// Mitsubishi GX Works2 project: 실린더제어ABAB   PLC: Q02/Q02H

PROGRAM MAIN
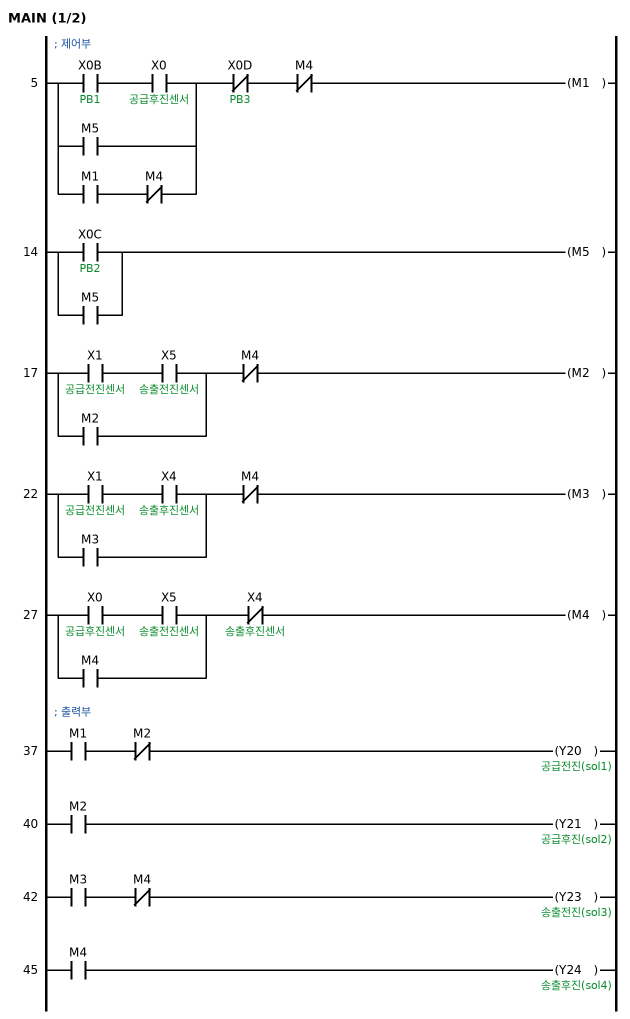
; 제어부
5     LD      X0B  ; PB1
      AND     X0  ; 공급후진센서
      OR      M5
      LD      M1
      ANI     M4
      ORB
      ANI     X0D  ; PB3
      ANI     M4
      OUT     M1
14    LD      X0C  ; PB2
      OR      M5
      OUT     M5
17    LD      X1  ; 공급전진센서
      AND     X5  ; 송출전진센서
      OR      M2
      ANI     M4
      OUT     M2
22    LD      X1  ; 공급전진센서
      AND     X4  ; 송출후진센서
      OR      M3
      ANI     M4
      OUT     M3
27    LD      X0  ; 공급후진센서
      AND     X5  ; 송출전진센서
      OR      M4
      ANI     X4  ; 송출후진센서
      OUT     M4
; 출력부
37    LD      M1
      ANI     M2
      OUT     Y20  ; 공급전진(sol1)
40    LD      M2
      OUT     Y21  ; 공급후진(sol2)
42    LD      M3
      ANI     M4
      OUT     Y23  ; 송출전진(sol3)
45    LD      M4
      OUT     Y24  ; 송출후진(sol4)
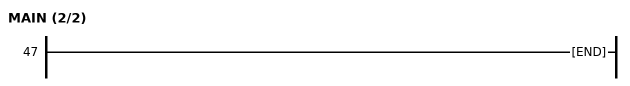
47    END
END_PROGRAM
